// TwinCAT 3 PLC project PLC
// ProgramVersion: 3.1.4022.3
// libraries:
//   Tc2_Standard, * (Beckhoff Automation GmbH)
//   Tc2_System, * (Beckhoff Automation GmbH)
//   Tc2_Utilities, * (Beckhoff Automation GmbH)
//   Tc3_Module, * (Beckhoff Automation GmbH)
// project tree:
//   DUTs/ Pancake.TcDUT
//   GVLs/ GVL.TcGVL
//   / PlcTask.TcTTO
//   POUs/ BottomUpMerge.TcPOU, CopyArray.TcPOU, MAIN.TcPOU, PanCakeBottomUpMergeSort.TcPOU, SolveChallenge.TcPOU
// real-time tasks:
//   TASK PlcTask: cycle T#1ms, priority 20, ADS port 350

CONFIGURATION PLC
    RESOURCE PLC ON TwinCAT3
        TASK PlcTask(INTERVAL := T#1ms, PRIORITY := 20);
        PROGRAM MAIN WITH PlcTask : MAIN;
    END_RESOURCE
END_CONFIGURATION

// ---- DUTs/Pancake.TcDUT
TYPE Pancake :
STRUCT
	Height:DINT;
	Radius:DINT;
	SideArea:LREAL;
	TotalArea:LREAL;
END_STRUCT
END_TYPE

// ---- GVLs/GVL.TcGVL
{attribute 'qualified_only'}
VAR_GLOBAL CONSTANT 
	MaxArraySize:INT:=999;	
END_VAR

// ---- POUs/MAIN.TcPOU
PROGRAM MAIN
VAR
	StartingTrigger:R_TRIG;	
	fbStringReader:FB_FileGets;
	fbFileOpener:FB_FileOpen;
	fbFileCloser:FB_FileClose;
	fbFileWriter:FB_FilePuts;
	State:INT;
	Execute:BOOL;
	T:INT; //Number of challenges
	N:INT; //Number of available pancakes
	K:INT; //Ordered pancakes
	Pancakes : ARRAY[0..GVL.MaxArraySize]  OF Pancake;  
	PancakeCounter:INT;
	ChallengeCounter:INT;
	Error:BOOL;
	ErrorCode:UDINT;
	SplitPosition:INT;
END_VAR

StartingTrigger(CLK:=Execute);
CASE State OF
	0: 	IF StartingTrigger.Q THEN
			State:=State+1;
			fbFileOpener.bExecute :=FALSE;
		END_IF
	 
	1:	fbFileOpener.sPathName :='C:\A-large-practice.in';
		fbFileOpener.nMode := FOPEN_MODEREAD;
		fbFileOpener.ePath := PATH_GENERIC;
		fbFileOpener(bExecute:=FALSE);
		fbFileOpener(bExecute:=TRUE);
		State:=State+1;
		
	2: 	fbFileOpener(bExecute:=FALSE);
		IF fbFileOpener.bError THEN
			State:=10;
			Error:=TRUE;
			ErrorCode:=fbFileOpener.nErrId;
		ELSIF NOT fbFileOpener.bBusy THEN			
			State:=State+1;
			fbStringReader.hFile := fbFileOpener.hFile;
			fbFileOpener.sPathName :='C:\Solution.out';
			fbFileOpener.nMode := FOPEN_MODEWRITE;
			fbFileOpener.ePath := PATH_GENERIC;			
			fbFileOpener(bExecute:=TRUE);
		END_IF  
 
	3: 	fbFileOpener(bExecute:=FALSE);
		IF fbFileOpener.bError THEN
			State:=10;
			Error:=TRUE;
			ErrorCode:=fbFileOpener.nErrId;
		ELSIF NOT fbFileOpener.bBusy THEN			
			State:=State+1;
			fbFileWriter.hFile := fbFileOpener.hFile;
		END_IF  
		
	4: 	fbStringReader.tTimeout:= T#1S;
		fbStringReader(bExecute := FALSE);
		fbStringReader(bExecute := TRUE );
		State:=State+1;
		
	5:  fbStringReader(bExecute := FALSE);
		IF fbStringReader.bError THEN
			State:=10;
			Error:=TRUE;
			ErrorCode:=fbStringReader.nErrId;
 		ELSIF NOT fbStringReader.bBusy THEN
			T := STRING_TO_INT(fbStringReader.sLine);
			ChallengeCounter :=0;
			fbStringReader(bExecute := TRUE);
			State:=State+1;
		END_IF
		
	6 : fbStringReader(bExecute := FALSE);
		IF fbStringReader.bError THEN
			State:=10;
			Error:=TRUE;
			ErrorCode:=fbStringReader.nErrId;
 		ELSIF NOT fbStringReader.bBusy THEN			
			SplitPosition := FIND(STR1:= fbStringReader.sLine, str2:= ' ');
			N:=STRING_TO_INT(LEFT(STR:=fbStringReader.sLine,SplitPosition));
			K:=STRING_TO_INT(MID(STR:=fbStringReader.sLine,LEN:= LEN(fbStringReader.sLine)-2,POS:=SplitPosition));	
			fbStringReader(bExecute := TRUE);
			State:=State+1;
			PancakeCounter :=0;
		END_IF	
		
	7 : fbStringReader(bExecute := FALSE);	
		IF fbStringReader.bError THEN
			State:=10;
			Error:=TRUE;
			ErrorCode:=fbStringReader.nErrId;
 		ELSIF NOT fbStringReader.bBusy THEN			
			SplitPosition := FIND(STR1:= fbStringReader.sLine, str2:= ' ');
			Pancakes[PancakeCounter].Radius:=STRING_TO_DINT(LEFT(STR:=fbStringReader.sLine,SplitPosition));
			Pancakes[PancakeCounter].Height:=STRING_TO_DINT(MID(STR:=fbStringReader.sLine,LEN:= LEN(fbStringReader.sLine)-2,POS:=SplitPosition));	
			Pancakes[PancakeCounter].SideArea:= 2*PI*Pancakes[PancakeCounter].Radius *Pancakes[PancakeCounter].Height;
			Pancakes[PancakeCounter].TotalArea :=PI *Pancakes[PancakeCounter].Radius *Pancakes[PancakeCounter].Radius +Pancakes[PancakeCounter].SideArea;
			PancakeCounter:=PancakeCounter+1;
			IF PancakeCounter = N THEN 
				State:=State+1;
			ELSE
				fbStringReader(bExecute := TRUE);	 
			END_IF
		END_IF		
		
	8:	fbFileWriter.sLine := CONCAT(CONCAT('Case #',INT_TO_STRING(ChallengeCounter+1)),': ');
		fbFileWriter.sLine := CONCAT(fbFileWriter.sLine,LREAL_TO_STRING(SolveChallenge(N:=N,K:=K,Pancakes:=Pancakes)));
		fbFileWriter.sLine := CONCAT(fbFileWriter.sLine,'$N');
		fbFileWriter.tTimeout :=T#1S;	
		fbFileWriter(bExecute:=FALSE);
		fbFileWriter(bExecute:=TRUE);		
		State:=State+1;
				
	9:	fbFileWriter(bExecute:=FALSE);
		IF NOT fbFileWriter.bBusy THEN 
			ChallengeCounter:= ChallengeCounter +1;
			IF ChallengeCounter < T THEN
				State:=6;
				fbStringReader(bExecute := TRUE);	 
			ELSE
				State:=State+1;
			END_IF			
		END_IF
		
	10: fbFileCloser.hFile := fbFileOpener.hFile;
		fbFileCloser.tTimeout :=T#1S;
		fbFileCloser(bExecute:=FALSE);
		fbFileCloser(bExecute:=TRUE);
		State:=State+1;
		
	11: fbFileCloser(bExecute:=FALSE);
		IF NOT fbFileCloser.bBusy THEN
			fbFileCloser.hFile := fbFileOpener.hFile;				
			fbFileCloser(bExecute:=TRUE);
			State:=State+1;
		END_IF
		
 	12: fbFileCloser(bExecute:=FALSE);
		IF NOT fbFileCloser.bBusy THEN										
			State:=0;
		END_IF
 END_CASE

END_PROGRAM

// ---- POUs/SolveChallenge.TcPOU
FUNCTION SolveChallenge : LREAL
VAR_INPUT
	N:INT; //Number of available pancakes
	K:INT; //Ordered pancakes
END_VAR
VAR_IN_OUT
	Pancakes : ARRAY[0..GVL.MaxArraySize]  OF Pancake; 
END_VAR
VAR
	i:INT;
	j:INT;
	PancakesBYSide : ARRAY[0..GVL.MaxArraySize]  OF Pancake; 
	WorkingArray : ARRAY[0..GVL.MaxArraySize]  OF Pancake; 
	StackArea:LREAL;
END_VAR

PanCakeBottomUpMergeSort(N:=N, SortBySideArea:=FALSE,ArrayToSort:=Pancakes, WorkingArray:=WorkingArray);

FOR i:=K-1 TO N-1 DO
	PancakesBYSide := Pancakes;
	StackArea :=Pancakes[i].TotalArea;
	PanCakeBottomUpMergeSort(N:=i, SortBySideArea:=TRUE,ArrayToSort:=PancakesBYSide , WorkingArray:=WorkingArray);
	FOR j:= 0 TO K-2 DO
		StackArea:= StackArea + PancakesBYSide[i-1 -j].SideArea;
	END_FOR
	SolveChallenge := MAX(SolveChallenge,StackArea);
END_FOR

END_FUNCTION

// ---- POUs/PanCakeBottomUpMergeSort.TcPOU
FUNCTION PanCakeBottomUpMergeSort
VAR_INPUT
	N:INT;//Number of elements
	SortBySideArea:BOOL; //True to sort the array by the side area of the pancakes. Other wise sort by radius
END_VAR
VAR_IN_OUT
	ArrayToSort: ARRAY[0..GVL.MaxArraySize]  OF Pancake;
	WorkingArray: ARRAY[0..GVL.MaxArraySize]  OF Pancake;
END_VAR
VAR 
	Width:INT;
	i:INT;
END_VAR

Width:=1;
WHILE (Width < N) DO
	i:=0;
	WHILE (i<N)DO
		BottomUpMerge(i,	MIN (i+Width,N),MIN(i+2*width, N),SortBySideArea,ArrayToSort,WorkingArray);
		i:=i+2*Width;
	END_WHILE
	CopyArray(N:=N,Source:= WorkingArray,Target:=ArrayToSort);	
	Width:= Width *2;
END_WHILE

END_FUNCTION

// ---- POUs/BottomUpMerge.TcPOU
FUNCTION BottomUpMerge
VAR_INPUT
	Left:INT;
	Right:INT;
	End:INT;
	SortBySideArea:BOOL;//True to sort the array by the side area of the pancakes. Other wise sort by radius
END_VAR
VAR_IN_OUT
	ArrayToSort: ARRAY[0..GVL.MaxArraySize]  OF Pancake;
	WorkingArray: ARRAY[0..GVL.MaxArraySize]  OF Pancake;
END_VAR
VAR
	i:INT;
	j:INT;
	k:INT;
END_VAR

i:=Left;
j:=Right;
FOR k:=left TO End DO
	IF (i<Right AND (j >=End OR 
			((NOT SortBySideArea AND ArrayToSort[i].Radius <=ArrayToSort[j].Radius) OR
			(SortBySideArea AND ArrayToSort[i].SideArea <=ArrayToSort[j].SideArea)))) THEN			
		WorkingArray[k] := ArrayToSort[i];
		i:=i+1;
	ELSE
		WorkingArray[k] := ArrayToSort[j];
		j:=j+1;
	END_IF
END_FOR

END_FUNCTION

// ---- POUs/CopyArray.TcPOU
FUNCTION CopyArray 
VAR_INPUT
	n:INT;	
END_VAR
VAR_IN_OUT
	Source: ARRAY[0..GVL.MaxArraySize]  OF Pancake;
	Target: ARRAY[0..GVL.MaxArraySize]  OF Pancake;
END_VAR
VAR
	i:INT;
END_VAR

FOR i:= 0 TO n DO
	Target[i]:=Source[i];
END_FOR

END_FUNCTION
